PROGRAM OperationPRG
VAR
	mxPosA 		  : BOOL;
	mxPosB 		  : BOOL;
	mxPosC 		  : BOOL;
	mxPosD 		  : BOOL;
	mxPosHome 	  : BOOL;
	mxPosInit 	  : BOOL;

END_VAR

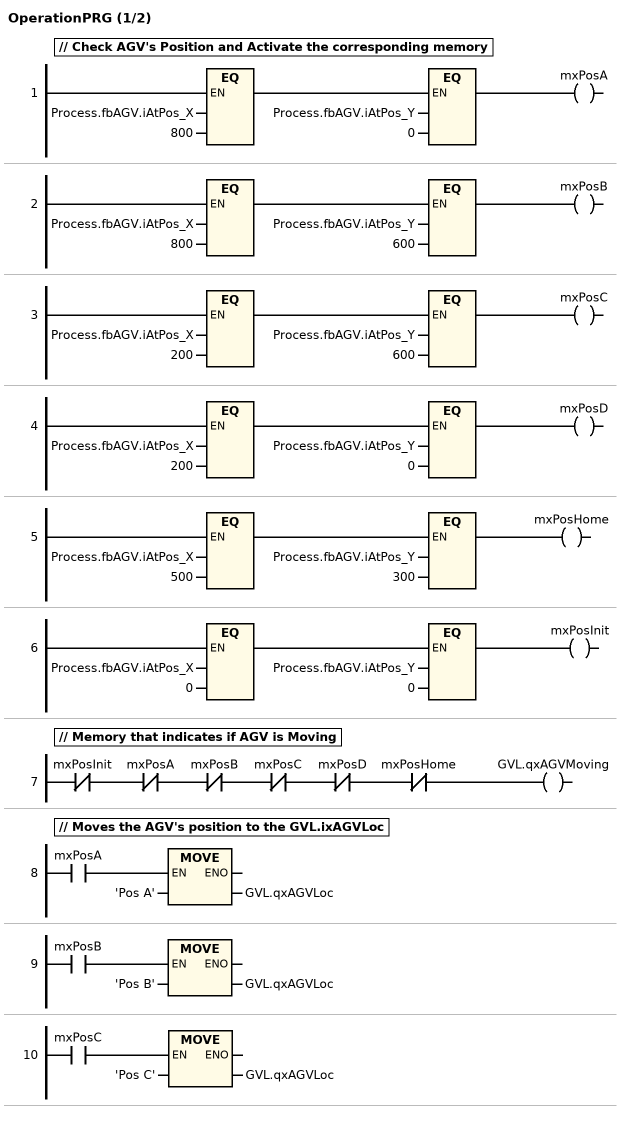
// NETWORK 1
// label: // Check AGV's Position and Activate the corresponding memory
mxPosA := Process.fbAGV.iAtPos_X = 800 AND Process.fbAGV.iAtPos_Y = 0;

// NETWORK 2
mxPosB := Process.fbAGV.iAtPos_X = 800 AND Process.fbAGV.iAtPos_Y = 600;

// NETWORK 3
mxPosC := Process.fbAGV.iAtPos_X = 200 AND Process.fbAGV.iAtPos_Y = 600;

// NETWORK 4
mxPosD := Process.fbAGV.iAtPos_X = 200 AND Process.fbAGV.iAtPos_Y = 0;

// NETWORK 5
mxPosHome := Process.fbAGV.iAtPos_X = 500 AND Process.fbAGV.iAtPos_Y = 300;

// NETWORK 6
mxPosInit := Process.fbAGV.iAtPos_X = 0 AND Process.fbAGV.iAtPos_Y = 0;

// NETWORK 7
// label: // Memory that indicates if AGV is Moving
GVL.qxAGVMoving := NOT mxPosInit AND NOT mxPosA AND NOT mxPosB AND NOT mxPosC AND NOT mxPosD AND NOT mxPosHome;

// NETWORK 8
// label: // Moves the AGV's position to the GVL.ixAGVLoc
IF mxPosA THEN GVL.qxAGVLoc := 'Pos A'; END_IF

// NETWORK 9
IF mxPosB THEN GVL.qxAGVLoc := 'Pos B'; END_IF

// NETWORK 10
IF mxPosC THEN GVL.qxAGVLoc := 'Pos C'; END_IF

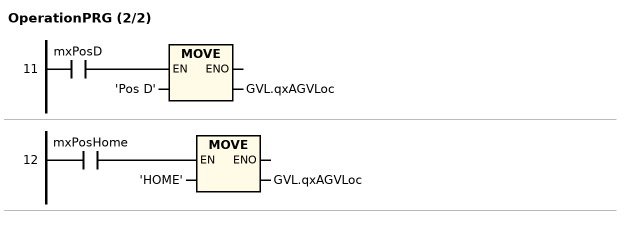
// NETWORK 11
IF mxPosD THEN GVL.qxAGVLoc := 'Pos D'; END_IF

// NETWORK 12
IF mxPosHome THEN GVL.qxAGVLoc := 'HOME'; END_IF

END_PROGRAM

(* stored: Version 1.1.0.1, ProductVersion 3.1.4024.12
   POU OperationPRG: Id {d7c66be7-90ee-41aa-ab2f-67b8319a3a7f}, SpecialFunc None *)
